PROGRAM example_loop_control
VAR
	//Example run request for a starter motor.  This would be triggered by control loop logic
	u_3160_a_run_request : BOOL;
	
	//Example run request for a vfd motor.  This would be triggered by control loop logic
	u_3112_a_run_request : BOOL;
	//Example Speed Request for a vfd motor.  This would be set by control loop logic, normally a PID
	u_3112_a_speed_request : REAL;
	
	//Example position request for an analog valve.  This would be set by control loop logic, normally a PID
	av_3148_a_position_request : REAL;
	
	//Example open request for a digital valve.  This would be triggered by control loop logic
	nv_3372_a_open_request : BOOL;
END_VAR

// NETWORK 1

END_PROGRAM

(* stored: Version 1.1.0.1, ProductVersion 3.1.4024.12
   POU example_loop_control: Id {f4111f27-f002-47e1-985a-deb6fca944d4}, SpecialFunc None *)
